// TIA Portal V15.1 export
// export: Created 2024-06-21T08:41:12.629283Z, ExportSetting WithDefaults, DisplayName Totally Integrated Automation Portal, DisplayVersion V15.1 Update 5, DisplayName TIA Portal Openness, DisplayVersion V15.1 Update 5, DisplayName SINAMICS Startdrive Advanced, DisplayVersion V15.1, DisplayName G130, G150, S120, S150, SINAMICS MV, S210, DisplayVersion V15.1, DisplayName G110M, G120, G120C, G120D, G120P, DisplayVersion V15.1, DisplayName STEP 7 Professional, DisplayVersion V15.1 Update 5, DisplayName STEP 7 Safety, DisplayVersion V15.1, DisplayName WinCC Professional, DisplayVersion V15.1 Update 5, DisplayName SIMATIC Visualization Architect, DisplayVersion V15.1
FUNCTION_BLOCK "LGBPassage"   // FB6681, FBD
TITLE = LGBPassage
{ S7_Optimized_Access := 'TRUE' }
VERSION : 0.1
// stored: AutoNumber false, IsIECCheckEnabled false, IsRetainMemResEnabled false, MemoryReserve 100, SetENOAutomatically False, UDAEnableTagReadback false
   VAR_INPUT
      I_ReqAccessStopPB { ExternalAccessible := 'False'; ExternalVisible := 'False'; ExternalWritable := 'False'} : Bool;   // Push button - Request for the pass through
      I_AcknowledgePB { ExternalAccessible := 'False'; ExternalVisible := 'False'; ExternalWritable := 'False'} : Bool;   // Push button - Acknowledge end of pass through
      I_AccessStopReached { ExternalAccessible := 'False'; ExternalVisible := 'False'; ExternalWritable := 'False'} : Bool;   // Request is Done for pass through
      I_EnableAlarm { ExternalAccessible := 'False'; ExternalVisible := 'False'; ExternalWritable := 'False'} : Bool := TRUE;   // Enable alarm from upper level / Enable Alarm from upper level
      I_SafetyOk { ExternalAccessible := 'False'; ExternalVisible := 'False'; ExternalWritable := 'False'} : Bool;   // Safety Passage SafetyOK
      I_InputGate1 { ExternalAccessible := 'False'; ExternalVisible := 'False'; ExternalWritable := 'False'} : Bool;
      I_AckReqGate1 { ExternalAccessible := 'False'; ExternalVisible := 'False'; ExternalWritable := 'False'} : Bool;
      I_InputGate2 { ExternalAccessible := 'False'; ExternalVisible := 'False'; ExternalWritable := 'False'} : Bool;
      I_AckReqGate2 { ExternalAccessible := 'False'; ExternalVisible := 'False'; ExternalWritable := 'False'} : Bool;
      I_InputScanner { ExternalAccessible := 'False'; ExternalVisible := 'False'; ExternalWritable := 'False'} : Bool;
      I_AckReqScanner { ExternalAccessible := 'False'; ExternalVisible := 'False'; ExternalWritable := 'False'} : Bool;
   END_VAR
   VAR_OUTPUT
      O_AccessStopReqSelected { ExternalAccessible := 'False'; ExternalVisible := 'False'; ExternalWritable := 'False'} : Bool;   // Access Stop Requested
      O_AccessStopReached { ExternalAccessible := 'False'; ExternalVisible := 'False'; ExternalWritable := 'False'} : Bool;   // Access Stop Reached/Ok to Cross
      O_AA_AccessedNotAllowed { ExternalAccessible := 'False'; ExternalVisible := 'False'; ExternalWritable := 'False'} : Bool;   // Accessed without Request
      O_AC_AccessOvertime { ExternalAccessible := 'False'; ExternalVisible := 'False'; ExternalWritable := 'False'} : Bool;
      O_AccessStopReq { ExternalAccessible := 'False'; ExternalVisible := 'False'; ExternalWritable := 'False'} : Bool;   // Warning when Access Requested (D)
      O_AlarmABCondition { ExternalAccessible := 'False'; ExternalVisible := 'False'; ExternalWritable := 'False'} : Bool;   // Alarm AB condition
      H_IAnim { ExternalAccessible := 'False'; ExternalVisible := 'False'; ExternalWritable := 'False'} : DWord;   // For animation of icon / Icon Animation
   END_VAR
   VAR_IN_OUT
      H_GBPassage : "H_GBPassage";   // Animation
   END_VAR
   VAR
      AccessReqSel { ExternalAccessible := 'False'; ExternalVisible := 'False'; ExternalWritable := 'False'} : Bool;   // Access Stop Requested
      AccessStopReached { ExternalAccessible := 'False'; ExternalVisible := 'False'; ExternalWritable := 'False'} : Bool;   // Access Stop Reached/Ok to Cross
      AccessOvertime { ExternalAccessible := 'False'; ExternalVisible := 'False'; ExternalWritable := 'False'} : Bool;   // Access Overtime
      _ToggleReqAccess { ExternalAccessible := 'False'; ExternalVisible := 'False'; ExternalWritable := 'False'} : "LToggle";
      Edge { ExternalAccessible := 'False'; ExternalVisible := 'False'; ExternalWritable := 'False'} : Array[1..4] of Bool;   // Edges / Edge
      TON_PassageOpen { ExternalAccessible := 'False'; ExternalVisible := 'False'; ExternalWritable := 'False'} : IEC_TIMER;
   END_VAR
   VAR_TEMP   // added for the SCL form of the ladder/FBD networks
      _w1 : Bool;
   END_VAR
BEGIN

REGION Network 1: *** 4.4 - Calculated **** Guard locking solenoid / **** 4.4 - Calculated **** Access Request Selected
   // Guard Locking Solenoid, Power to unlock (True = unlocked / False = locked) / Guard Locking Solenoid (True = locked / False = unlocked) / Access Request Selected
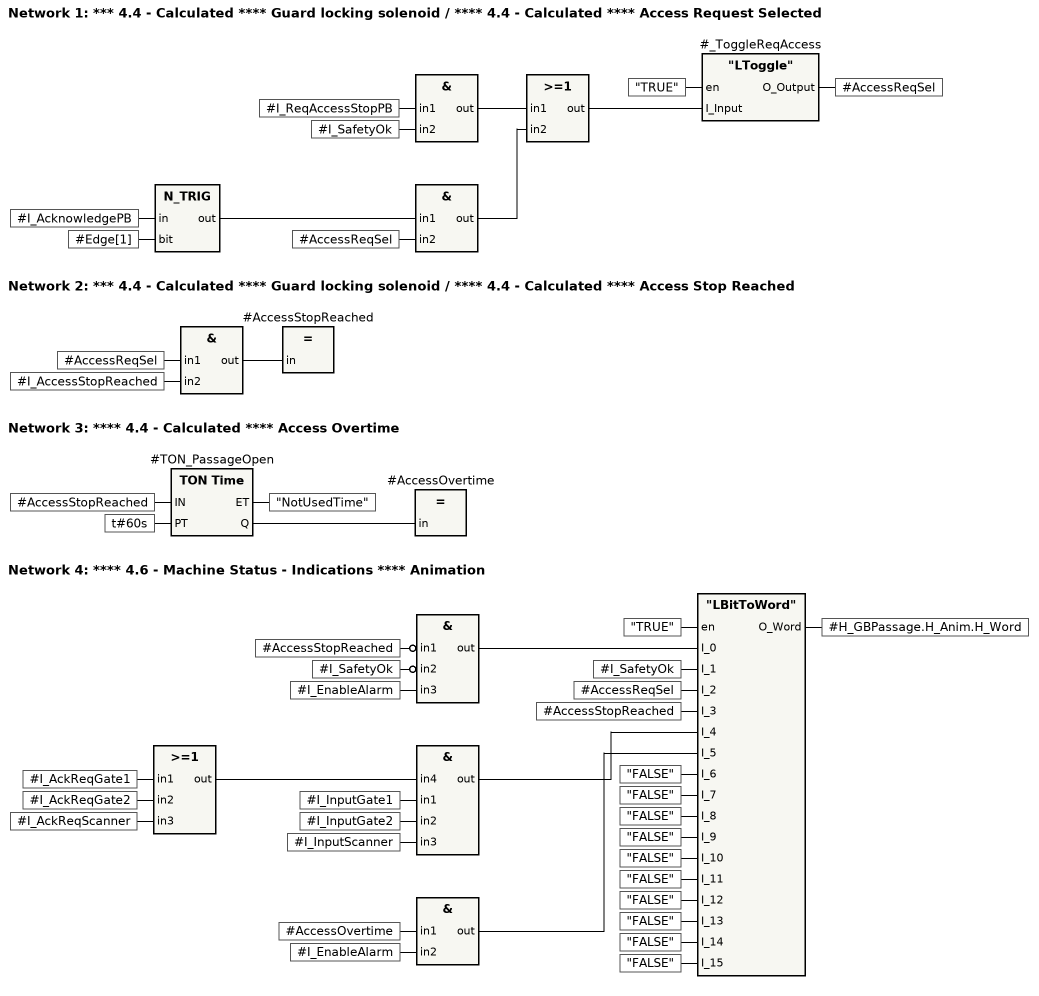
   #_w1 := NOT #I_AcknowledgePB AND #Edge[1];   // falling edge
   #Edge[1] := #I_AcknowledgePB;
   IF "TRUE" THEN
       #_ToggleReqAccess(I_Input := (#I_ReqAccessStopPB AND #I_SafetyOk) OR (#_w1 AND #AccessReqSel),   // "LToggle"
                         O_Output => #AccessReqSel);
   END_IF;
END_REGION

REGION Network 2: *** 4.4 - Calculated **** Guard locking solenoid / **** 4.4 - Calculated **** Access Stop Reached
   // Guard Locking Solenoid, Power to unlock (True = unlocked / False = locked) / Guard Locking Solenoid (True = locked / False = unlocked) / Access Stop Reached
   #AccessStopReached := #AccessReqSel AND #I_AccessStopReached;
END_REGION

REGION Network 3: **** 4.4 - Calculated **** Access Overtime
   // 60s passed from requesting time
   #TON_PassageOpen.TON(IN := #AccessStopReached, PT := t#60s, ET => "NotUsedTime");
   #AccessOvertime := #TON_PassageOpen.Q;
END_REGION

REGION Network 4: **** 4.6 - Machine Status - Indications **** Animation
   // Animation
   IF "TRUE" THEN
       "LBitToWord"(I_0 := NOT #AccessStopReached AND NOT #I_SafetyOk AND #I_EnableAlarm,
                    I_1 := #I_SafetyOk,
                    I_2 := #AccessReqSel,
                    I_3 := #AccessStopReached,
                    I_4 := (#I_AckReqGate1 OR #I_AckReqGate2 OR #I_AckReqScanner) AND #I_InputGate1 AND #I_InputGate2 AND #I_InputScanner,
                    I_5 := #AccessOvertime AND #I_EnableAlarm,
                    I_6 := "FALSE",
                    I_7 := "FALSE",
                    I_8 := "FALSE",
                    I_9 := "FALSE",
                    I_10 := "FALSE",
                    I_11 := "FALSE",
                    I_12 := "FALSE",
                    I_13 := "FALSE",
                    I_14 := "FALSE",
                    I_15 := "FALSE",
                    O_Word => #H_GBPassage.H_Anim.H_Word);
   END_IF;
END_REGION

REGION Network 5: **** 4.6 - Machine Status - Indication **** Icon Animation
   // Icon Animation for HMI
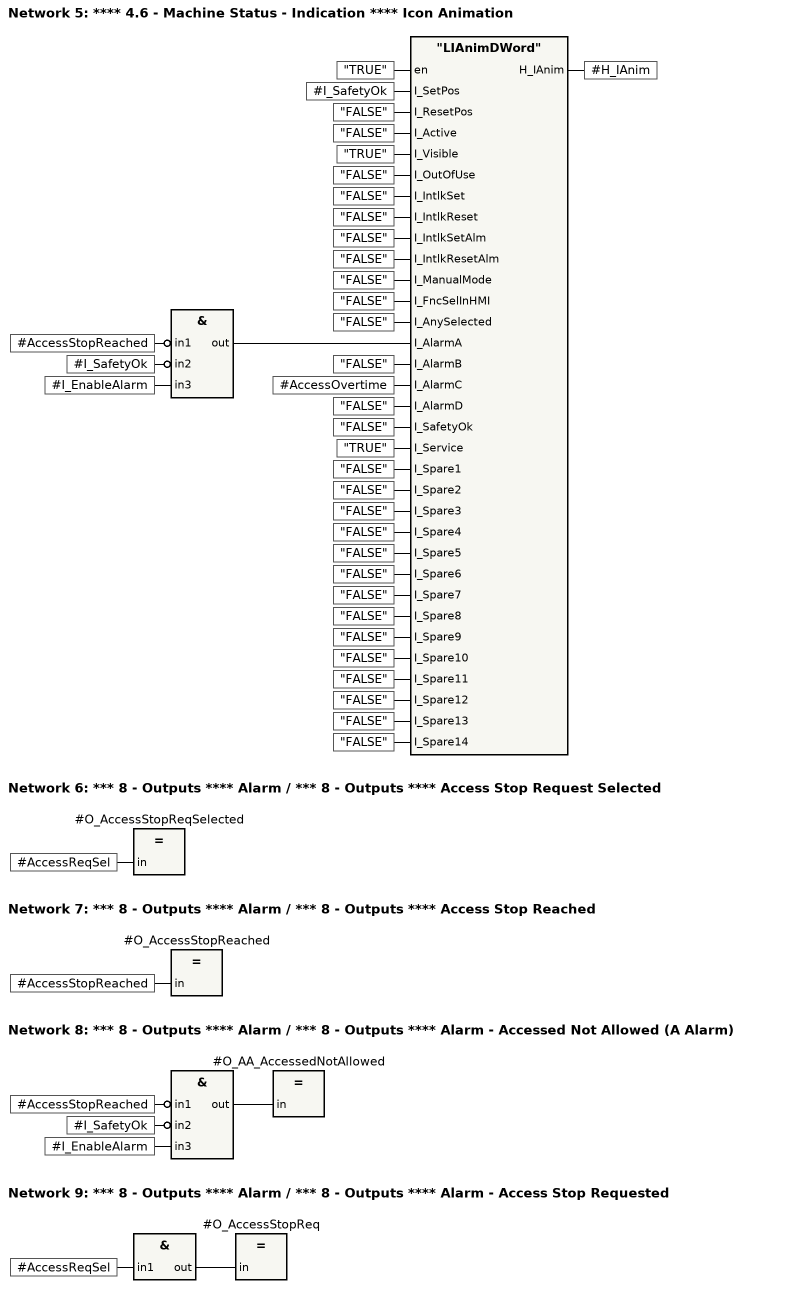
   IF "TRUE" THEN
       "LIAnimDWord"(I_SetPos := #I_SafetyOk,
                     I_ResetPos := "FALSE",
                     I_Active := "FALSE",
                     I_Visible := "TRUE",
                     I_OutOfUse := "FALSE",
                     I_IntlkSet := "FALSE",
                     I_IntlkReset := "FALSE",
                     I_IntlkSetAlm := "FALSE",
                     I_IntlkResetAlm := "FALSE",
                     I_ManualMode := "FALSE",
                     I_FncSelInHMI := "FALSE",
                     I_AnySelected := "FALSE",
                     I_AlarmA := NOT #AccessStopReached AND NOT #I_SafetyOk AND #I_EnableAlarm,
                     I_AlarmB := "FALSE",
                     I_AlarmC := #AccessOvertime,
                     I_AlarmD := "FALSE",
                     I_SafetyOk := "FALSE",
                     I_Service := "TRUE",
                     I_Spare1 := "FALSE",
                     I_Spare2 := "FALSE",
                     I_Spare3 := "FALSE",
                     I_Spare4 := "FALSE",
                     I_Spare5 := "FALSE",
                     I_Spare6 := "FALSE",
                     I_Spare7 := "FALSE",
                     I_Spare8 := "FALSE",
                     I_Spare9 := "FALSE",
                     I_Spare10 := "FALSE",
                     I_Spare11 := "FALSE",
                     I_Spare12 := "FALSE",
                     I_Spare13 := "FALSE",
                     I_Spare14 := "FALSE",
                     H_IAnim => #H_IAnim);
   END_IF;
END_REGION

REGION Network 6: *** 8 - Outputs **** Alarm / *** 8 - Outputs **** Access Stop Request Selected
   // Output Of The Alarm / Access Stop Request Selected
   #O_AccessStopReqSelected := #AccessReqSel;
END_REGION

REGION Network 7: *** 8 - Outputs **** Alarm / *** 8 - Outputs **** Access Stop Reached
   // Output Of The Alarm / Access Allowed
   #O_AccessStopReached := #AccessStopReached;
END_REGION

REGION Network 8: *** 8 - Outputs **** Alarm / *** 8 - Outputs **** Alarm - Accessed Not Allowed (A Alarm)
   // Output Of The Alarm / Alarm - Crossing without Access Request
   #O_AA_AccessedNotAllowed := NOT #AccessStopReached AND NOT #I_SafetyOk AND #I_EnableAlarm;
END_REGION

REGION Network 9: *** 8 - Outputs **** Alarm / *** 8 - Outputs **** Alarm - Access Stop Requested
   // Output Of The Alarm / AccessReqSel
   #O_AccessStopReq := #AccessReqSel;
END_REGION

REGION Network 10: *** 8 - Outputs **** Alarm - Access Stop Overtime (C Warning)
   // Overtime
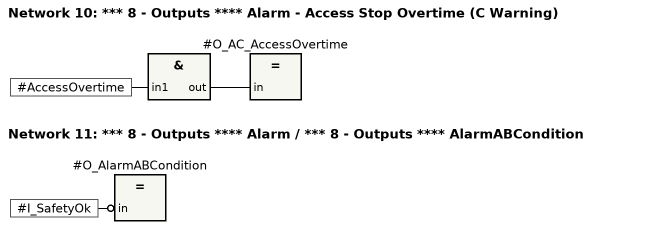
   #O_AC_AccessOvertime := #AccessOvertime;
END_REGION

REGION Network 11: *** 8 - Outputs **** Alarm / *** 8 - Outputs **** AlarmABCondition
   // Output Of The Alarm / AlarmABCondition
   #O_AlarmABCondition := NOT #I_SafetyOk;
END_REGION
END_FUNCTION_BLOCK
